// TIA Portal V19 export
VAR_GLOBAL   // PLC tag table "Mémoires"
   "Hauteur (pourcentage)" AT %MD0 : Real;   // Valeur de la hauteur de la pièce en pourcentage
   "Activer Q1" AT %M4.0 : Bool;   // Mémoire pour activer Q1
   "Mémoire compteur noires" AT %M4.1 : Bool;   // Mémoire pour les fronts montants du cpt noires
   "Mémoire compteur mauvaise hauteur" AT %M4.2 : Bool;   // Mémoire pour les fronts montants du cpt mauvaises pièces
   "Mémoire compteur bonne hauteur" AT %M4.3 : Bool;   // Mémoire pour les fronts montants du cpt bonnes pièces
   "Clock 1Hz" AT %M250.5 : Bool;
   "Clock 2Hz" AT %M250.3 : Bool;
   "Clock 0,625Hz" AT %M250.6 : Bool;
   "Clock 0,5Hz" AT %M250.7 : Bool;
   "Clock 1,5Hz" AT %M250.4 : Bool;
   "Clock 2,5Hz" AT %M250.2 : Bool;
   "Clock 5Hz" AT %M250.1 : Bool;
   "Clock 10Hz" AT %M250.0 : Bool;
   RETVAL_WWW AT %MW80 : Int;
   Start_Stop AT %M10.0 : Bool;
   Compteur AT %MW2 : Int;
   PieceMax AT %MW100 : Int;
   "Compteur Bonnes Pièces" AT %MW10 : Int;
   "Compteur Mauvaises Pièces" AT %MW12 : Int;
   "Pointeur 1" AT %MD50 : DWord;
   "Pointeur 2" AT %MD54 : DWord;
   "A CHANGER" AT %MW200 : Word;
   "NB Bonnes Pièces" AT %MW26 : Word;   // Nombre des bonnes pièces à afficher sur le web serveur
   "NB Mauvaises Pièces" AT %MW28 : Word;   // Nombre des mauvaises pièces à afficher sur le web serveur
   BPStartWeb AT %M251.0 : Bool;
   BPStopWeb AT %M251.1 : Bool;
   BPResetWeb AT %M251.2 : Bool;
   TestMax AT %M251.3 : Bool;
   BoolDeResetMauvaisePiece AT %MW70 : Int;
   BoolDeResetBonnePiece AT %MW72 : Int;
END_VAR
